// TIA Portal project "Module 1 PLC" (V16)

(* hardware
DEVICE "S7-1200 station_2"  S7-1200 Station
   slot 0: "Rack_0"  S7-1200 Rack  Rack  V1.0
   slot 1: "PLC_2"  CPU 1214C DC/DC/DC  6ES7 214-1AG40-0XB0  V4.0
   slot 2: "DI 8/DQ 8x24VDC_1"  SM 1223 DI8/DQ8 x 24VDC  6ES7 223-1BH30-0XB0  V1.0
*)

// ===== PLC "PLC_2"  CPU 1214C DC/DC/DC =====

VAR_GLOBAL   // PLC tag table "Default tag table"
   "Tag_1" AT %M20.5 : Bool;
END_VAR

VAR_GLOBAL   // PLC tag table "Default tag table_1"
   "System_Byte" AT %MB100 : Byte;
   "FirstScan" AT %M100.0 : Bool;
   "DiagStatusUpdate" AT %M100.1 : Bool;
   "AlwaysTRUE" AT %M100.2 : Bool;
   "AlwaysFALSE" AT %M100.3 : Bool;
   "Clock_Byte" AT %MB200 : Byte;
   "Clock_10Hz" AT %M200.0 : Bool;
   "Clock_5Hz" AT %M200.1 : Bool;
   "Clock_2.5Hz" AT %M200.2 : Bool;
   "Clock_2Hz" AT %M200.3 : Bool;
   "Clock_1.25Hz" AT %M200.4 : Bool;
   "Clock_1Hz" AT %M200.5 : Bool;
   "Clock_0.625Hz" AT %M200.6 : Bool;
   "Clock_0.5Hz" AT %M200.7 : Bool;
   "START" AT %I0.0 : Bool;
   "STOP" AT %I0.1 : Bool;
   "RESET" AT %I0.2 : Bool;
   "CBD" AT %I0.3 : Bool;
   "CBC" AT %I0.6 : Bool;
   "CBP" AT %I2.1 : Bool;
   "S1AC" AT %I0.7 : Bool;
   "S1AD" AT %I2.0 : Bool;
   "S2AT" AT %I2.6 : Bool;
   "S2AP" AT %I2.4 : Bool;
   "S3AX" AT %I2.2 : Bool;
   "S3AL" AT %I2.3 : Bool;
   "S4AX" AT %I0.4 : Bool;
   "S4AL" AT %I0.5 : Bool;
   "S2AG" AT %I2.5 : Bool;
   "ST1" AT %M0.0 : Bool;
   "ST2" AT %M0.1 : Bool;
   "ST3" AT %M0.2 : Bool;
   "ST4" AT %M0.3 : Bool;
   "ST5" AT %M0.4 : Bool;
   "ST6" AT %M0.5 : Bool;
   "ST7" AT %M0.6 : Bool;
   "ST8" AT %M0.7 : Bool;
   "ST9" AT %M1.0 : Bool;
   "ST10" AT %M1.1 : Bool;
   "ST11" AT %M1.2 : Bool;
   "ST12" AT %M1.3 : Bool;
   "ST13" AT %M1.4 : Bool;
   "ST14" AT %M1.5 : Bool;
   "ST15" AT %M1.6 : Bool;
   "ST16" AT %M1.7 : Bool;
   "ST17" AT %M2.0 : Bool;
   "ST18" AT %M2.1 : Bool;
   "K1AD" AT %Q0.5 : Bool;
   "K2AT" AT %Q1.1 : Bool;
   "K2AP" AT %Q0.2 : Bool;
   "K3AX" AT %Q0.3 : Bool;
   "K4AX" AT %Q0.0 : Bool;
   "BT" AT %Q2.0 : Bool;
   "GH" AT %Q0.4 : Bool;
   "R" AT %Q2.1 : Bool;
   "Y" AT %Q2.3 : Bool;
   "G" AT %Q2.2 : Bool;
   "Tag_1(1)" AT %M20.0 : Bool;
   "Tag_2(1)" AT %M10.0 : Bool;
   "CBPL" AT %I2.7 : Bool;
END_VAR

VAR_GLOBAL CONSTANT   // PLC tag table "Default tag table_1"
   "None(1)" : Pip := 65535;
   "Automatic update(1)" : Pip := 0;
   "PIP 1(1)" : Pip := 1;
   "PIP 2(1)" : Pip := 2;
   "PIP 3(1)" : Pip := 3;
   "PIP 4(1)" : Pip := 4;
   "PIP OB Servo(1)" : Pip := 32768;
   "Local~Exec(1)" : Hw_SubModule := 52;
   "Local(1)" : Hw_SubModule := 49;
   "Local~PROFINET_interface_1~Port_1(1)" : Hw_Interface := 65;
   "Local~AI_2_1(1)" : Hw_SubModule := 263;
   "OB_Main(1)" : OB_PCYCLE := 1;
   "Local~DI_8_DQ_8x24VDC_1(1)" : Hw_SubModule := 269;
   "Local~DI_14_DQ_10_1(1)" : Hw_SubModule := 257;
   "Local~MC(1)" : Hw_SubModule := 51;
   "Local~Common(1)" : Hw_SubModule := 50;
   "Local~Pulse_1(1)" : Hw_Pwm := 258;
   "Local~Pulse_2(1)" : Hw_Pwm := 259;
   "Local~Pulse_3(1)" : Hw_Pwm := 260;
   "Local~Pulse_4(1)" : Hw_Pwm := 261;
   "Local~PROFINET_interface_1(1)" : Hw_Interface := 64;
   "Local~HSC_1(1)" : Hw_Hsc := 262;
   "Local~HSC_2(1)" : Hw_Hsc := 264;
   "Local~HSC_3(1)" : Hw_Hsc := 265;
   "Local~HSC_4(1)" : Hw_Hsc := 266;
   "Local~HSC_5(1)" : Hw_Hsc := 267;
   "Local~HSC_6(1)" : Hw_Hsc := 268;
END_VAR

// folder: System blocks/Program resources

DATA_BLOCK "T1"   // DB1
{ S7_Optimized_Access := 'TRUE' }
AUTHOR : Simatic
FAMILY : IEC
NAME : IEC_TMR
VERSION : 1.0
// stored: InstanceOfName IEC_TIMER
"IEC_TIMER"
BEGIN
END_DATA_BLOCK

DATA_BLOCK "T2"   // DB2
{ S7_Optimized_Access := 'TRUE' }
AUTHOR : Simatic
FAMILY : IEC
NAME : IEC_TMR
VERSION : 1.0
// stored: InstanceOfName IEC_TIMER
"IEC_TIMER"
BEGIN
END_DATA_BLOCK

DATA_BLOCK "T5"   // DB3
{ S7_Optimized_Access := 'TRUE' }
AUTHOR : Simatic
FAMILY : IEC
NAME : IEC_TMR
VERSION : 1.0
// stored: InstanceOfName IEC_TIMER
"IEC_TIMER"
BEGIN
END_DATA_BLOCK

DATA_BLOCK "T3"   // DB4
{ S7_Optimized_Access := 'TRUE' }
AUTHOR : Simatic
FAMILY : IEC
NAME : IEC_TMR
VERSION : 1.0
// stored: InstanceOfName IEC_TIMER
"IEC_TIMER"
BEGIN
END_DATA_BLOCK

DATA_BLOCK "T4"   // DB5
{ S7_Optimized_Access := 'TRUE' }
AUTHOR : Simatic
FAMILY : IEC
NAME : IEC_TMR
VERSION : 1.0
// stored: InstanceOfName IEC_TIMER
"IEC_TIMER"
BEGIN
END_DATA_BLOCK

// folder: (top level)

ORGANIZATION_BLOCK "Main"   // OB1, LAD, ProgramCycle
TITLE = "Main Program Sweep (Cycle)"
{ S7_Optimized_Access := 'TRUE' }
VERSION : 0.1
   VAR_INPUT
      Initial_Call : Bool;   // Initial call of this OB
      Remanence : Bool;   // =True, if remanent data are available
   END_VAR
BEGIN

REGION Network 1
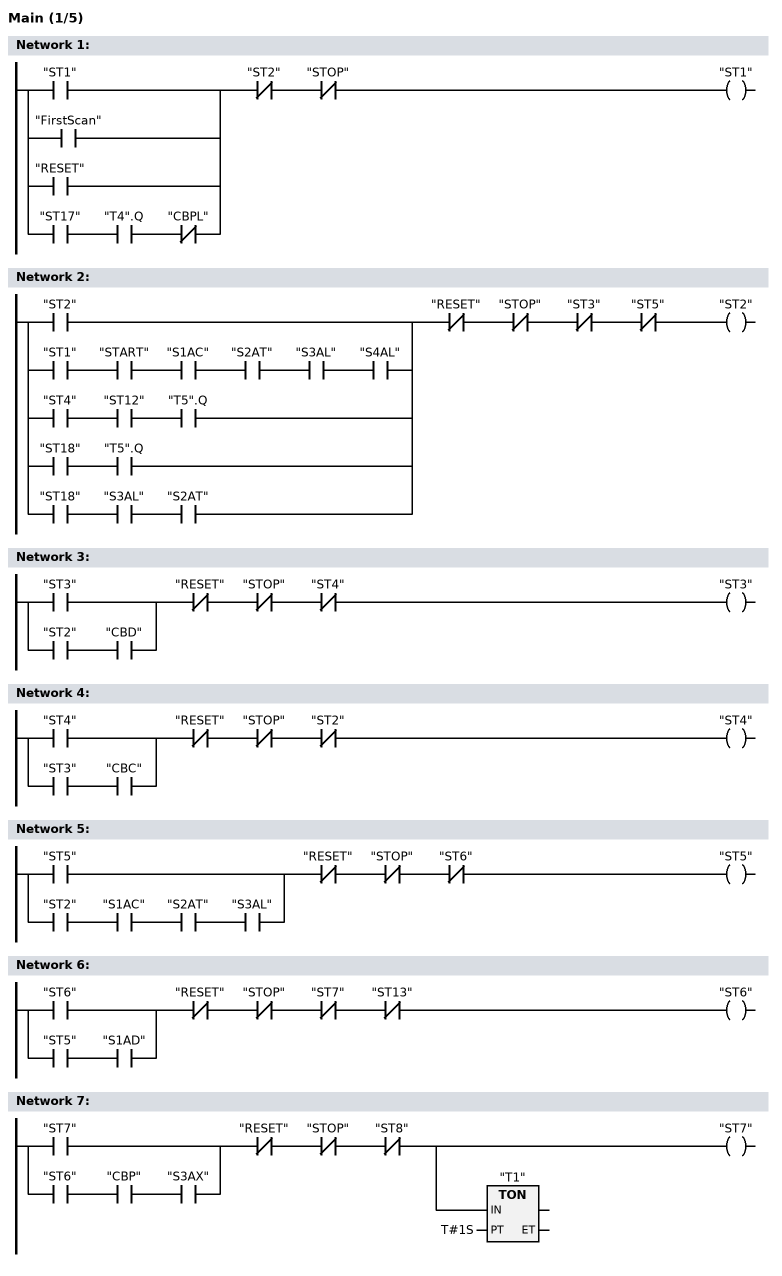
   RUNG wire#powerrail
      Contact( "ST1" )
      wire#w1
      I_Contact( "ST2" )
      I_Contact( "STOP" )
      Coil( "ST1" )
   END_RUNG
   RUNG wire#powerrail
      Contact( "FirstScan" )
   END_RUNG wire#w1
   RUNG wire#powerrail
      Contact( "RESET" )
   END_RUNG wire#w1
   RUNG wire#powerrail
      Contact( "ST17" )
      Contact( "T4".Q )
      I_Contact( "CBPL" )
   END_RUNG wire#w1
   // the same network as SCL:
   "ST1" := ("ST1" OR "FirstScan" OR "RESET" OR ("ST17" AND "T4".Q AND NOT "CBPL")) AND NOT "ST2" AND NOT "STOP";
END_REGION

REGION Network 2
   RUNG wire#powerrail
      Contact( "ST2" )
      wire#w1
      I_Contact( "RESET" )
      I_Contact( "STOP" )
      I_Contact( "ST3" )
      I_Contact( "ST5" )
      Coil( "ST2" )
   END_RUNG
   RUNG wire#powerrail
      Contact( "ST1" )
      Contact( "START" )
      Contact( "S1AC" )
      Contact( "S2AT" )
      Contact( "S3AL" )
      Contact( "S4AL" )
   END_RUNG wire#w1
   RUNG wire#powerrail
      Contact( "ST4" )
      Contact( "ST12" )
      Contact( "T5".Q )
   END_RUNG wire#w1
   RUNG wire#powerrail
      Contact( "ST18" )
      Contact( "T5".Q )
   END_RUNG wire#w1
   RUNG wire#powerrail
      Contact( "ST18" )
      Contact( "S3AL" )
      Contact( "S2AT" )
   END_RUNG wire#w1
   // the same network as SCL:
   "ST2" := ("ST2" OR ("ST1" AND "START" AND "S1AC" AND "S2AT" AND "S3AL" AND "S4AL") OR ("ST4" AND "ST12" AND "T5".Q) OR ("ST18" AND "T5".Q) OR ("ST18" AND "S3AL" AND "S2AT")) AND NOT "RESET" AND NOT "STOP" AND NOT "ST3" AND NOT "ST5";
END_REGION

REGION Network 3
   RUNG wire#powerrail
      Contact( "ST3" )
      wire#w1
      I_Contact( "RESET" )
      I_Contact( "STOP" )
      I_Contact( "ST4" )
      Coil( "ST3" )
   END_RUNG
   RUNG wire#powerrail
      Contact( "ST2" )
      Contact( "CBD" )
   END_RUNG wire#w1
   // the same network as SCL:
   "ST3" := ("ST3" OR ("ST2" AND "CBD")) AND NOT "RESET" AND NOT "STOP" AND NOT "ST4";
END_REGION

REGION Network 4
   RUNG wire#powerrail
      Contact( "ST4" )
      wire#w1
      I_Contact( "RESET" )
      I_Contact( "STOP" )
      I_Contact( "ST2" )
      Coil( "ST4" )
   END_RUNG
   RUNG wire#powerrail
      Contact( "ST3" )
      Contact( "CBC" )
   END_RUNG wire#w1
   // the same network as SCL:
   "ST4" := ("ST4" OR ("ST3" AND "CBC")) AND NOT "RESET" AND NOT "STOP" AND NOT "ST2";
END_REGION

REGION Network 5
   RUNG wire#powerrail
      Contact( "ST5" )
      wire#w1
      I_Contact( "RESET" )
      I_Contact( "STOP" )
      I_Contact( "ST6" )
      Coil( "ST5" )
   END_RUNG
   RUNG wire#powerrail
      Contact( "ST2" )
      Contact( "S1AC" )
      Contact( "S2AT" )
      Contact( "S3AL" )
   END_RUNG wire#w1
   // the same network as SCL:
   "ST5" := ("ST5" OR ("ST2" AND "S1AC" AND "S2AT" AND "S3AL")) AND NOT "RESET" AND NOT "STOP" AND NOT "ST6";
END_REGION

REGION Network 6
   RUNG wire#powerrail
      Contact( "ST6" )
      wire#w1
      I_Contact( "RESET" )
      I_Contact( "STOP" )
      I_Contact( "ST7" )
      I_Contact( "ST13" )
      Coil( "ST6" )
   END_RUNG
   RUNG wire#powerrail
      Contact( "ST5" )
      Contact( "S1AD" )
   END_RUNG wire#w1
   // the same network as SCL:
   "ST6" := ("ST6" OR ("ST5" AND "S1AD")) AND NOT "RESET" AND NOT "STOP" AND NOT "ST7" AND NOT "ST13";
END_REGION

REGION Network 7
   "ST7" := ("ST7" OR ("ST6" AND "CBP" AND "S3AX")) AND NOT "RESET" AND NOT "STOP" AND NOT "ST8";
   "T1".TON(IN := "ST7", PT := T#1S);
END_REGION

REGION Network 8
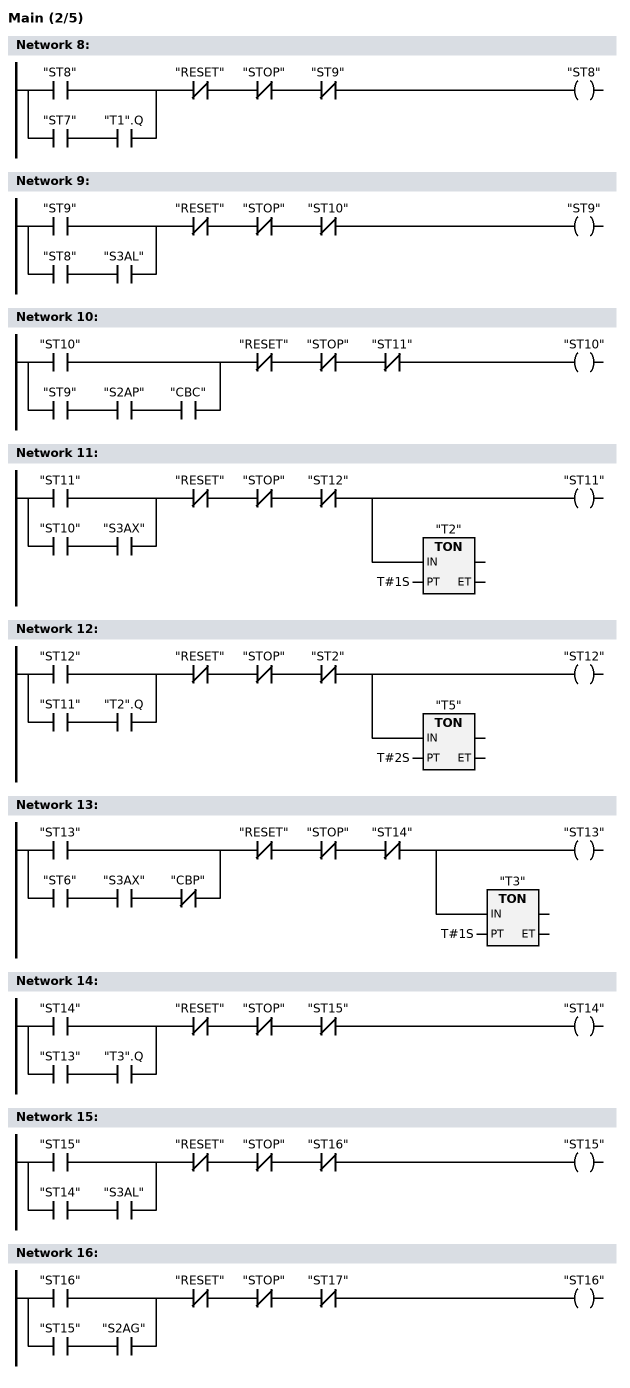
   RUNG wire#powerrail
      Contact( "ST8" )
      wire#w1
      I_Contact( "RESET" )
      I_Contact( "STOP" )
      I_Contact( "ST9" )
      Coil( "ST8" )
   END_RUNG
   RUNG wire#powerrail
      Contact( "ST7" )
      Contact( "T1".Q )
   END_RUNG wire#w1
   // the same network as SCL:
   "ST8" := ("ST8" OR ("ST7" AND "T1".Q)) AND NOT "RESET" AND NOT "STOP" AND NOT "ST9";
END_REGION

REGION Network 9
   RUNG wire#powerrail
      Contact( "ST9" )
      wire#w1
      I_Contact( "RESET" )
      I_Contact( "STOP" )
      I_Contact( "ST10" )
      Coil( "ST9" )
   END_RUNG
   RUNG wire#powerrail
      Contact( "ST8" )
      Contact( "S3AL" )
   END_RUNG wire#w1
   // the same network as SCL:
   "ST9" := ("ST9" OR ("ST8" AND "S3AL")) AND NOT "RESET" AND NOT "STOP" AND NOT "ST10";
END_REGION

REGION Network 10
   RUNG wire#powerrail
      Contact( "ST10" )
      wire#w1
      I_Contact( "RESET" )
      I_Contact( "STOP" )
      I_Contact( "ST11" )
      Coil( "ST10" )
   END_RUNG
   RUNG wire#powerrail
      Contact( "ST9" )
      Contact( "S2AP" )
      Contact( "CBC" )
   END_RUNG wire#w1
   // the same network as SCL:
   "ST10" := ("ST10" OR ("ST9" AND "S2AP" AND "CBC")) AND NOT "RESET" AND NOT "STOP" AND NOT "ST11";
END_REGION

REGION Network 11
   "ST11" := ("ST11" OR ("ST10" AND "S3AX")) AND NOT "RESET" AND NOT "STOP" AND NOT "ST12";
   "T2".TON(IN := "ST11", PT := T#1S);
END_REGION

REGION Network 12
   "ST12" := ("ST12" OR ("ST11" AND "T2".Q)) AND NOT "RESET" AND NOT "STOP" AND NOT "ST2";
   "T5".TON(IN := "ST12", PT := T#2S);
END_REGION

REGION Network 13
   "ST13" := ("ST13" OR ("ST6" AND "S3AX" AND NOT "CBP")) AND NOT "RESET" AND NOT "STOP" AND NOT "ST14";
   "T3".TON(IN := "ST13", PT := T#1S);
END_REGION

REGION Network 14
   RUNG wire#powerrail
      Contact( "ST14" )
      wire#w1
      I_Contact( "RESET" )
      I_Contact( "STOP" )
      I_Contact( "ST15" )
      Coil( "ST14" )
   END_RUNG
   RUNG wire#powerrail
      Contact( "ST13" )
      Contact( "T3".Q )
   END_RUNG wire#w1
   // the same network as SCL:
   "ST14" := ("ST14" OR ("ST13" AND "T3".Q)) AND NOT "RESET" AND NOT "STOP" AND NOT "ST15";
END_REGION

REGION Network 15
   RUNG wire#powerrail
      Contact( "ST15" )
      wire#w1
      I_Contact( "RESET" )
      I_Contact( "STOP" )
      I_Contact( "ST16" )
      Coil( "ST15" )
   END_RUNG
   RUNG wire#powerrail
      Contact( "ST14" )
      Contact( "S3AL" )
   END_RUNG wire#w1
   // the same network as SCL:
   "ST15" := ("ST15" OR ("ST14" AND "S3AL")) AND NOT "RESET" AND NOT "STOP" AND NOT "ST16";
END_REGION

REGION Network 16
   RUNG wire#powerrail
      Contact( "ST16" )
      wire#w1
      I_Contact( "RESET" )
      I_Contact( "STOP" )
      I_Contact( "ST17" )
      Coil( "ST16" )
   END_RUNG
   RUNG wire#powerrail
      Contact( "ST15" )
      Contact( "S2AG" )
   END_RUNG wire#w1
   // the same network as SCL:
   "ST16" := ("ST16" OR ("ST15" AND "S2AG")) AND NOT "RESET" AND NOT "STOP" AND NOT "ST17";
END_REGION

REGION Network 17
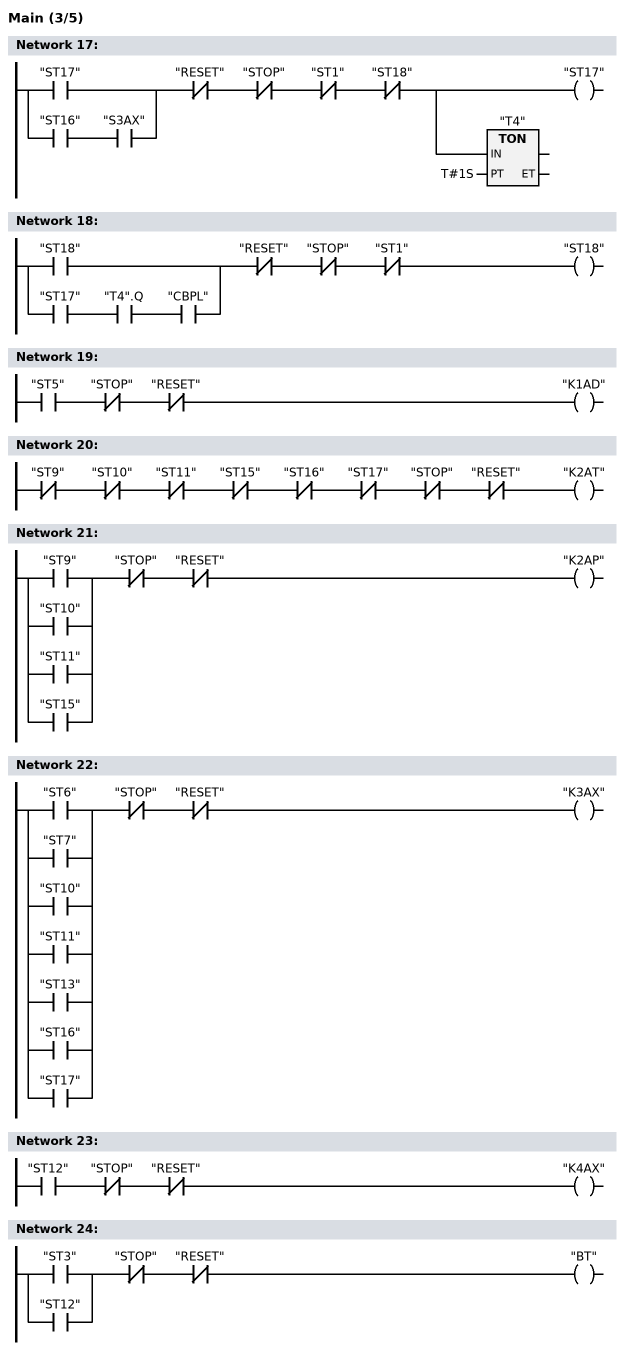
   "ST17" := ("ST17" OR ("ST16" AND "S3AX")) AND NOT "RESET" AND NOT "STOP" AND NOT "ST1" AND NOT "ST18";
   "T4".TON(IN := "ST17", PT := T#1S);
END_REGION

REGION Network 18
   RUNG wire#powerrail
      Contact( "ST18" )
      wire#w1
      I_Contact( "RESET" )
      I_Contact( "STOP" )
      I_Contact( "ST1" )
      Coil( "ST18" )
   END_RUNG
   RUNG wire#powerrail
      Contact( "ST17" )
      Contact( "T4".Q )
      Contact( "CBPL" )
   END_RUNG wire#w1
   // the same network as SCL:
   "ST18" := ("ST18" OR ("ST17" AND "T4".Q AND "CBPL")) AND NOT "RESET" AND NOT "STOP" AND NOT "ST1";
END_REGION

REGION Network 19
   RUNG wire#powerrail
      Contact( "ST5" )
      I_Contact( "STOP" )
      I_Contact( "RESET" )
      Coil( "K1AD" )
   END_RUNG
   // the same network as SCL:
   "K1AD" := "ST5" AND NOT "STOP" AND NOT "RESET";
END_REGION

REGION Network 20
   RUNG wire#powerrail
      I_Contact( "ST9" )
      I_Contact( "ST10" )
      I_Contact( "ST11" )
      I_Contact( "ST15" )
      I_Contact( "ST16" )
      I_Contact( "ST17" )
      I_Contact( "STOP" )
      I_Contact( "RESET" )
      Coil( "K2AT" )
   END_RUNG
   // the same network as SCL:
   "K2AT" := NOT "ST9" AND NOT "ST10" AND NOT "ST11" AND NOT "ST15" AND NOT "ST16" AND NOT "ST17" AND NOT "STOP" AND NOT "RESET";
END_REGION

REGION Network 21
   RUNG wire#powerrail
      Contact( "ST9" )
      wire#w1
      I_Contact( "STOP" )
      I_Contact( "RESET" )
      Coil( "K2AP" )
   END_RUNG
   RUNG wire#powerrail
      Contact( "ST10" )
   END_RUNG wire#w1
   RUNG wire#powerrail
      Contact( "ST11" )
   END_RUNG wire#w1
   RUNG wire#powerrail
      Contact( "ST15" )
   END_RUNG wire#w1
   // the same network as SCL:
   "K2AP" := ("ST9" OR "ST10" OR "ST11" OR "ST15") AND NOT "STOP" AND NOT "RESET";
END_REGION

REGION Network 22
   RUNG wire#powerrail
      Contact( "ST6" )
      wire#w1
      I_Contact( "STOP" )
      I_Contact( "RESET" )
      Coil( "K3AX" )
   END_RUNG
   RUNG wire#powerrail
      Contact( "ST7" )
   END_RUNG wire#w1
   RUNG wire#powerrail
      Contact( "ST10" )
   END_RUNG wire#w1
   RUNG wire#powerrail
      Contact( "ST11" )
   END_RUNG wire#w1
   RUNG wire#powerrail
      Contact( "ST13" )
   END_RUNG wire#w1
   RUNG wire#powerrail
      Contact( "ST16" )
   END_RUNG wire#w1
   RUNG wire#powerrail
      Contact( "ST17" )
   END_RUNG wire#w1
   // the same network as SCL:
   "K3AX" := ("ST6" OR "ST7" OR "ST10" OR "ST11" OR "ST13" OR "ST16" OR "ST17") AND NOT "STOP" AND NOT "RESET";
END_REGION

REGION Network 23
   RUNG wire#powerrail
      Contact( "ST12" )
      I_Contact( "STOP" )
      I_Contact( "RESET" )
      Coil( "K4AX" )
   END_RUNG
   // the same network as SCL:
   "K4AX" := "ST12" AND NOT "STOP" AND NOT "RESET";
END_REGION

REGION Network 24
   RUNG wire#powerrail
      Contact( "ST3" )
      wire#w1
      I_Contact( "STOP" )
      I_Contact( "RESET" )
      Coil( "BT" )
   END_RUNG
   RUNG wire#powerrail
      Contact( "ST12" )
   END_RUNG wire#w1
   // the same network as SCL:
   "BT" := ("ST3" OR "ST12") AND NOT "STOP" AND NOT "RESET";
END_REGION

REGION Network 25
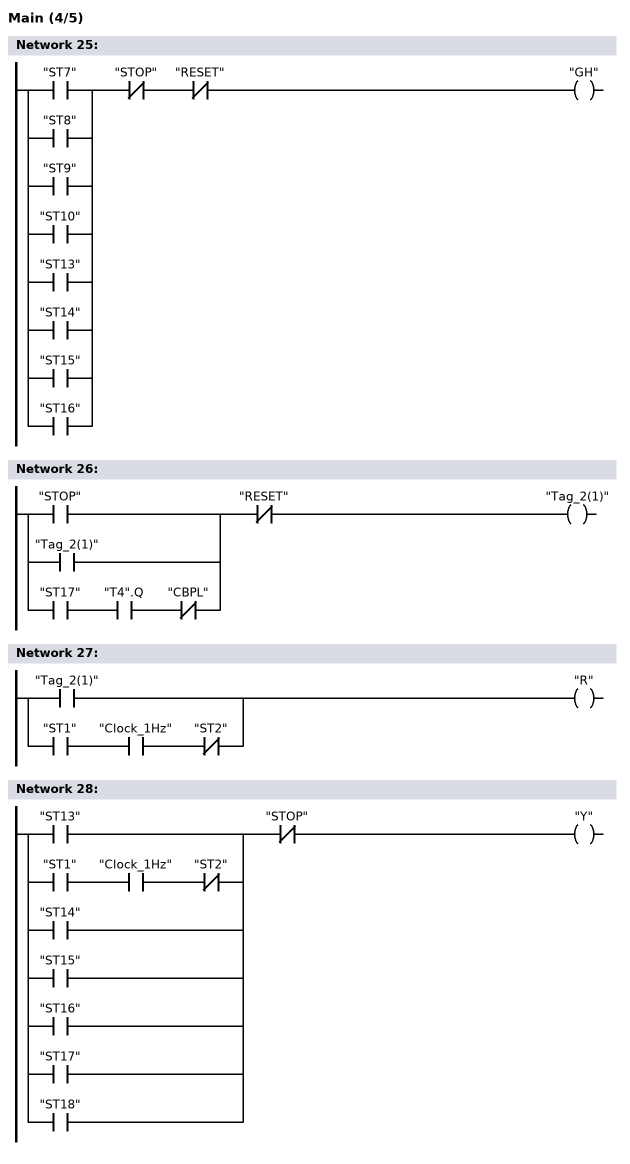
   RUNG wire#powerrail
      Contact( "ST7" )
      wire#w1
      I_Contact( "STOP" )
      I_Contact( "RESET" )
      Coil( "GH" )
   END_RUNG
   RUNG wire#powerrail
      Contact( "ST8" )
   END_RUNG wire#w1
   RUNG wire#powerrail
      Contact( "ST9" )
   END_RUNG wire#w1
   RUNG wire#powerrail
      Contact( "ST10" )
   END_RUNG wire#w1
   RUNG wire#powerrail
      Contact( "ST13" )
   END_RUNG wire#w1
   RUNG wire#powerrail
      Contact( "ST14" )
   END_RUNG wire#w1
   RUNG wire#powerrail
      Contact( "ST15" )
   END_RUNG wire#w1
   RUNG wire#powerrail
      Contact( "ST16" )
   END_RUNG wire#w1
   // the same network as SCL:
   "GH" := ("ST7" OR "ST8" OR "ST9" OR "ST10" OR "ST13" OR "ST14" OR "ST15" OR "ST16") AND NOT "STOP" AND NOT "RESET";
END_REGION

REGION Network 26
   RUNG wire#powerrail
      Contact( "STOP" )
      wire#w1
      I_Contact( "RESET" )
      Coil( "Tag_2(1)" )
   END_RUNG
   RUNG wire#powerrail
      Contact( "Tag_2(1)" )
   END_RUNG wire#w1
   RUNG wire#powerrail
      Contact( "ST17" )
      Contact( "T4".Q )
      I_Contact( "CBPL" )
   END_RUNG wire#w1
   // the same network as SCL:
   "Tag_2(1)" := ("STOP" OR "Tag_2(1)" OR ("ST17" AND "T4".Q AND NOT "CBPL")) AND NOT "RESET";
END_REGION

REGION Network 27
   RUNG wire#powerrail
      Contact( "Tag_2(1)" )
      wire#w1
      Coil( "R" )
   END_RUNG
   RUNG wire#powerrail
      Contact( "ST1" )
      Contact( "Clock_1Hz" )
      I_Contact( "ST2" )
   END_RUNG wire#w1
   // the same network as SCL:
   "R" := "Tag_2(1)" OR ("ST1" AND "Clock_1Hz" AND NOT "ST2");
END_REGION

REGION Network 28
   RUNG wire#powerrail
      Contact( "ST13" )
      wire#w1
      I_Contact( "STOP" )
      Coil( "Y" )
   END_RUNG
   RUNG wire#powerrail
      Contact( "ST1" )
      Contact( "Clock_1Hz" )
      I_Contact( "ST2" )
   END_RUNG wire#w1
   RUNG wire#powerrail
      Contact( "ST14" )
   END_RUNG wire#w1
   RUNG wire#powerrail
      Contact( "ST15" )
   END_RUNG wire#w1
   RUNG wire#powerrail
      Contact( "ST16" )
   END_RUNG wire#w1
   RUNG wire#powerrail
      Contact( "ST17" )
   END_RUNG wire#w1
   RUNG wire#powerrail
      Contact( "ST18" )
   END_RUNG wire#w1
   // the same network as SCL:
   "Y" := ("ST13" OR ("ST1" AND "Clock_1Hz" AND NOT "ST2") OR "ST14" OR "ST15" OR "ST16" OR "ST17" OR "ST18") AND NOT "STOP";
END_REGION

REGION Network 29
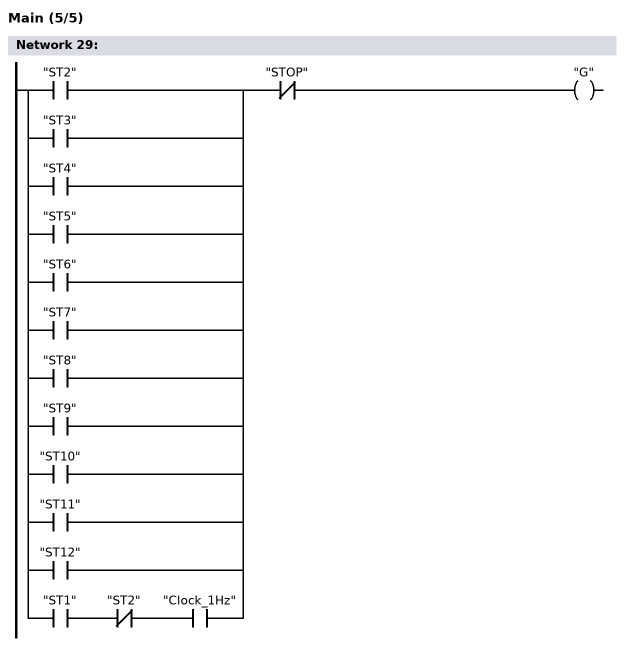
   RUNG wire#powerrail
      Contact( "ST2" )
      wire#w1
      I_Contact( "STOP" )
      Coil( "G" )
   END_RUNG
   RUNG wire#powerrail
      Contact( "ST3" )
   END_RUNG wire#w1
   RUNG wire#powerrail
      Contact( "ST4" )
   END_RUNG wire#w1
   RUNG wire#powerrail
      Contact( "ST5" )
   END_RUNG wire#w1
   RUNG wire#powerrail
      Contact( "ST6" )
   END_RUNG wire#w1
   RUNG wire#powerrail
      Contact( "ST7" )
   END_RUNG wire#w1
   RUNG wire#powerrail
      Contact( "ST8" )
   END_RUNG wire#w1
   RUNG wire#powerrail
      Contact( "ST9" )
   END_RUNG wire#w1
   RUNG wire#powerrail
      Contact( "ST10" )
   END_RUNG wire#w1
   RUNG wire#powerrail
      Contact( "ST11" )
   END_RUNG wire#w1
   RUNG wire#powerrail
      Contact( "ST12" )
   END_RUNG wire#w1
   RUNG wire#powerrail
      Contact( "ST1" )
      I_Contact( "ST2" )
      Contact( "Clock_1Hz" )
   END_RUNG wire#w1
   // the same network as SCL:
   "G" := ("ST2" OR "ST3" OR "ST4" OR "ST5" OR "ST6" OR "ST7" OR "ST8" OR "ST9" OR "ST10" OR "ST11" OR "ST12" OR ("ST1" AND NOT "ST2" AND "Clock_1Hz")) AND NOT "STOP";
END_REGION
END_ORGANIZATION_BLOCK